(*

## Short summary

This interface provides assert statements for signed integers from 8~64 bit length 
For 8 bit intgers use `ISignedIntegerAssertions.short`
For 16 bit intgers use `ISignedIntegerAssertions.simple`
For 32 bit intgers use `ISignedIntegerAssertions.double`
For 64 bit intgers use `ISignedIntegerAssertions.long`
For integers in register length use `ISignedIntegerAssertions.x`

.. <legal notes>

legal notes
=================
| SPDX-FileCopyrightText: © 2022 ekvip automation GmbH <info@ekvip.de>
| SPDX-License-Identifier: Apache-2.0
| For details check: Apache-2.0_

.. _Apache-2.0: https://www.apache.org/licenses/LICENSE-2.0

.. </legal notes>

properties
==================

*)

INTERFACE ISignedIntegerAssertions EXTENDS __SYSTEM.IQueryInterface

(*

## Short summary
Returns the interface `IDintAssertions` with assert statements for signed 32 bit integers 

.. <legal notes>

legal notes
=================
| SPDX-FileCopyrightText: © 2022 ekvip automation GmbH <info@ekvip.de>
| SPDX-License-Identifier: Apache-2.0
| For details check: Apache-2.0_

.. _Apache-2.0: https://www.apache.org/licenses/LICENSE-2.0

.. </legal notes>

*)

PROPERTY double :IDintAssertions
GET
END_GET
END_PROPERTY

(*

## Short summary
Returns the interface `ILintAssertions` with assert statements for signed 64 bit integers 

.. <legal notes>

legal notes
=================
| SPDX-FileCopyrightText: © 2022 ekvip automation GmbH <info@ekvip.de>
| SPDX-License-Identifier: Apache-2.0
| For details check: Apache-2.0_

.. _Apache-2.0: https://www.apache.org/licenses/LICENSE-2.0

.. </legal notes>

*)

PROPERTY long :ILintAssertions
GET
END_GET
END_PROPERTY

(*

## Short summary
Returns the interface `ISintAssertions` with assert statements for signed 8 bit integers 

.. <legal notes>

legal notes
=================
| SPDX-FileCopyrightText: © 2022 ekvip automation GmbH <info@ekvip.de>
| SPDX-License-Identifier: Apache-2.0
| For details check: Apache-2.0_

.. _Apache-2.0: https://www.apache.org/licenses/LICENSE-2.0

.. </legal notes>

*)

PROPERTY short :ISintAssertions
GET
END_GET
END_PROPERTY

(*

## Short summary
Returns the interface `IIntAssertions` with assert statements for signed 16 bit integers 

.. <legal notes>

legal notes
=================
| SPDX-FileCopyrightText: © 2022 ekvip automation GmbH <info@ekvip.de>
| SPDX-License-Identifier: Apache-2.0
| For details check: Apache-2.0_

.. _Apache-2.0: https://www.apache.org/licenses/LICENSE-2.0

.. </legal notes>

*)

PROPERTY simple :IIntAssertions
GET
END_GET
END_PROPERTY

(*

## Short summary
Returns the interface `IXintAssertions` with assert statements for signed integers register length 

.. <legal notes>

legal notes
=================
| SPDX-FileCopyrightText: © 2022 ekvip automation GmbH <info@ekvip.de>
| SPDX-License-Identifier: Apache-2.0
| For details check: Apache-2.0_

.. _Apache-2.0: https://www.apache.org/licenses/LICENSE-2.0

.. </legal notes>

*)

PROPERTY x :IXintAssertions
GET
END_GET
END_PROPERTY

END_INTERFACE

(* stored: Version 1.1.0.1, ProductVersion 3.1.4024.11
   Itf ISignedIntegerAssertions: Id {637cd7b1-41f2-4b19-8a1e-cab47c68c582}
   Property double: Id {eaa89ec6-67c0-4acf-93ed-bf061ae0dcda}
   Get Get: Id {f90905b3-e1d1-4c26-af57-2323cc2f254d}
   Property long: Id {32faab82-2192-4a5c-9379-e7a7e1550021}
   Get Get: Id {8765439c-2184-417d-837b-50873ffa56f1}
   Property short: Id {e292d4f4-824f-4b0c-8ad9-2c519f616974}
   Get Get: Id {2baa5923-a252-4a03-badc-c12e6b539013}
   Property simple: Id {aa0ed2ee-99b7-4e2a-ab3b-d51308b5c3da}
   Get Get: Id {70a64b33-1a36-4a65-a8c1-4d56e64402c3}
   Property x: Id {7a1fb43c-5930-4a28-b9e1-ddcc56932764}
   Get Get: Id {0f089141-cc88-4563-be61-addb9a5c72db} *)
